PROGRAM MAIN
VAR
itest :INT;
END_VAR

END_PROGRAM

(* stored: Version 1.1.0.1, ProductVersion 3.1.0.36
   POU MAIN: Id {1d3502ef-77da-4b8c-9d82-c1494c626a2b} *)
